TYPE "MEStoPLC_ST350_ext"
VERSION : 0.1
   STRUCT
      MainCheckIn : "MEStoPLC_MainCheckIn_ext";
      SubCheckIn : "MEStoPLC_SubCheckIn_ext";
      ScanResultsStored : "MEStoPLC_ResultsStoredScanExchange_ext";
      MarkingPrintExchange : "MEStoPLC_PrintExchange_ext";
      MainCheckOut : "MEStoPLC_MainCheckOut_ext";
      Common : "MEStoPLC_Common_ext";
   END_STRUCT;

END_TYPE

